Fanuc KAREL source: kt00049.KL

-- PROVISIONAL review KL for V770-1; original PC SHA256 93271043f0e7a8be7ab2008df44ae9563be4fe7dd5ac6d3444408ddec7a213a2
-- Incomplete behavior may be omitted. Consult companion uncertainty JSON. Do not deploy.
PROGRAM KT00049
%NOLOCKGROUP
VAR
  I2 : INTEGER
  OUT : INTEGER
-- UNRESOLVED_DECL Y1 type=002018
BEGIN
  -- UNRESOLVED_PC offsets 5-19; opcodes 2E,22,9D,33,B2
  -- UNRESOLVED_PC offsets 24-35; opcodes 2E,23
  -- UNRESOLVED_PC offsets 40-62; opcodes 22,9D,33,B1,21,53,23
  -- UNRESOLVED_PC offsets 67-71; opcodes 7F
END KT00049
